(* CoDeSys 2.3.9.47 project: gym_err.prx *)
(* Libraries: TcBaseBX.lbx 10.5.06 08:50:20, TcSystemBX.lbx 11.6.12 13:56:16, standard.lbx 5.12.03 08:02:30, TcEIB.lbx 16.5.14 14:12:22, TcBABasicBX.lbx 22.7.15 15:46:56 *)

(* Task configuration *)
TASK Standard (PRIORITY := 0, INTERVAL := T#20ms);
	MAIN
END_TASK

(* Global variable list: Global_Variables *)
VAR_GLOBAL
END_VAR

VAR_GLOBAL RETAIN
	eib_gym01:							 BOOL;
	eib_gym02:							 BOOL;
	eib_training01:						 BOOL;
	eib_training02:						 BOOL;
	eib_training03	:						 BOOL;
	eib_gym_stairs_bra:					 BOOL;
	eib_pool_hall_spotlight:				 BOOL;
	eib_pool_hall_LED:					 BOOL;

	eib_pool_light:						 BOOL;
	eib_sphere_ceiling_light:				 BOOL;
	eib_sphere_light:						 BOOL;
	eib_sphere_stars_light:					 BOOL;
	eib_gym_shower01_light:				 BOOL;
	eib_gym_shower02_light:				 BOOL;
	eib_gym_WC_corridor:					 BOOL;
	eib_gym_stairs_light:					 BOOL;

	eib_gym_WC_light:					 BOOL;
	eib_training:							 BOOL;
	eib_gym:								 BOOL;

	eib_training_1column_light	:			BOOL;
	eib_pool_inwater	:					BOOL;

	eib_pool_floor_heating_pump:			BOOL := TRUE ;
	eib_gym_floor_heating_pump:			BOOL := TRUE;
	eib_vent_heating_pump:				BOOL := TRUE;
	eib_heating_pump:					BOOL := TRUE;

	eib_outside_bigBulbs:					 BOOL;
	eib_outside_pingPongTable:			 BOOL;
	eib_outside_plantsLightning:			 BOOL;
	eib_outside_smallBulbs:				 BOOL;
END_VAR

(* Global variable list: KNX *)
VAR_GLOBAL
	fb_KL6301_0:								KL6301;


	fb_gym01_send_status_ex: 					EIB_BIT_SEND_EX;
	fb_gym02_send_status_ex: 					EIB_BIT_SEND_EX;
	fb_training01_send_status_ex: 				EIB_BIT_SEND_EX;
	fb_training02_send_status_ex: 				EIB_BIT_SEND_EX;
	fb_training03_send_status_ex: 				EIB_BIT_SEND_EX;
	fb_gym_stairs_bra_send_status_ex: 			EIB_BIT_SEND_EX;
	fb_pool_hall_spotlight_send_status_ex: 		EIB_BIT_SEND_EX;
	fb_pool_hall_LED_send_status_ex: 			EIB_BIT_SEND_EX;

	fb_pool_light_send_status_ex: 				EIB_BIT_SEND_EX;
	fb_sphere_ceiling_light_send_status_ex: 		EIB_BIT_SEND_EX;
	fb_sphere_light_send_status_ex: 			EIB_BIT_SEND_EX;
	fb_sphere_stars_light_send_status_ex: 		EIB_BIT_SEND_EX;
	fb_gym_shower01_light_send_status_ex: 		EIB_BIT_SEND_EX;
	fb_gym_shower02_light_send_status_ex: 		EIB_BIT_SEND_EX;
	fb_gym_WC_corridor_send_status_ex: 		EIB_BIT_SEND_EX;
	fb_gym_stairs_light_send_status_ex: 			EIB_BIT_SEND_EX;

	fb_gym_WC_light_send_status_ex: 			EIB_BIT_SEND_EX;
	fb_training_light_send_status_ex: 			EIB_BIT_SEND_EX;
	fb_gym_light_send_status_ex: 				EIB_BIT_SEND_EX;

	fb_gym_all_send_status_ex: 				EIB_BIT_SEND_EX;
	fb_training_all_send_status_ex: 				EIB_BIT_SEND_EX;
	fb_training_1column_send_status_ex: 		EIB_BIT_SEND_EX;
	fb_pool_inwater_send_status_ex: 			EIB_BIT_SEND_EX;


	fb_outside_bigBulbs_send_status_ex:		EIB_BIT_SEND_EX;
	fb_outside_smallBulbs_send_status_ex:		EIB_BIT_SEND_EX;
	fb_outside_pingPongTable_send_status_ex:	EIB_BIT_SEND_EX;
	fb_outside_plantsLightning_send_status_ex:	EIB_BIT_SEND_EX;

	fb_pool_floor_heating_pump_send_status_ex:	EIB_BIT_SEND_EX;
	fb_gym_floor_heating_pump_send_status_ex:	EIB_BIT_SEND_EX;
	fb_vent_heating_pump_send_status_ex:		EIB_BIT_SEND_EX;
	fb_heating_pump_send_status_ex:			EIB_BIT_SEND_EX;


	fb_pool_floor_heating_pump_read:			EIB_BIT_REC ;
	fb_gym_floor_heating_pump_read:			EIB_BIT_REC ;
	fb_vent_heating_pump_read:				EIB_BIT_REC ;
	fb_heating_pump_read:					EIB_BIT_REC ;

	fb_gym01_read: 					EIB_BIT_REC;
	fb_gym02_read: 					EIB_BIT_REC;
	fb_training01_read:				EIB_BIT_REC;
	fb_training02_read:				EIB_BIT_REC;
	fb_training03_read:				EIB_BIT_REC;
	fb_gym_stairs_bra_read:			EIB_BIT_REC;
	fb_pool_hall_spotlight_read:		EIB_BIT_REC;
	fb_pool_hall_LED_read:			EIB_BIT_REC;

	fb_pool_light_read:				EIB_BIT_REC;
	fb_sphere_ceiling_light_read:		EIB_BIT_REC;
	fb_sphere_light_read:				EIB_BIT_REC;
	fb_sphere_stars_light_read:			EIB_BIT_REC;
	fb_gym_shower01_light_read:		EIB_BIT_REC;
	fb_gym_shower02_light_read:		EIB_BIT_REC;
	fb_gym_WC_corridor_read:			EIB_BIT_REC;
	fb_gym_stairs_light_read:			EIB_BIT_REC;

	fb_gym_WC_light_read:			EIB_BIT_REC;
	fb_training_light_read:				EIB_BIT_REC;
	fb_gym_light_read:				EIB_BIT_REC;
	fb_outside_bigBulbs_read:			EIB_BIT_REC;
	fb_outside_smallBulbs_read:		EIB_BIT_REC;
	fb_outside_pingPongTable_read:	EIB_BIT_REC;
	fb_outside_plantsLightning_read:	EIB_BIT_REC;

	fb_gym_all_read: 					EIB_BIT_REC;
	fb_training_all_read: 				EIB_BIT_REC;
	fb_training_1column_read: 			EIB_BIT_REC;
	fb_pool_inwater_read: 				EIB_BIT_REC;

	gym_lights					:	BOOL;


(*2/0/x*)
	pool_floor_heating_pump_adr:								EIB_GROUP_ADDR :=(MAIN:=2, SUB_MAIN:=0, NUMBER:=1);
	gym_floor_heating_pump_adr:								EIB_GROUP_ADDR :=(MAIN:=2, SUB_MAIN:=0, NUMBER:=2);
	vent_heating_pump_adr:									EIB_GROUP_ADDR :=(MAIN:=2, SUB_MAIN:=0, NUMBER:=3);
	heating_pump_adr:										EIB_GROUP_ADDR :=(MAIN:=2, SUB_MAIN:=0, NUMBER:=4);

	pool_floor_heating_pump_status_adr:						EIB_GROUP_ADDR :=(MAIN:=2, SUB_MAIN:=0, NUMBER:=101);
	gym_floor_heating_pump_status_adr:							EIB_GROUP_ADDR :=(MAIN:=2, SUB_MAIN:=0, NUMBER:=102);
	vent_heating_pump_status_adr:								EIB_GROUP_ADDR :=(MAIN:=2, SUB_MAIN:=0, NUMBER:=103);
	heating_pump_staus_adr:									EIB_GROUP_ADDR :=(MAIN:=2, SUB_MAIN:=0, NUMBER:=104);


(*2/1/x*)
	gym01_adr:												EIB_GROUP_ADDR :=(MAIN:=2, SUB_MAIN:=1, NUMBER:=1);
	gym02_adr:												EIB_GROUP_ADDR :=(MAIN:=2, SUB_MAIN:=1, NUMBER:=2);
	training01_adr:											EIB_GROUP_ADDR :=(MAIN:=2, SUB_MAIN:=1, NUMBER:=3);
	training02_adr:											EIB_GROUP_ADDR :=(MAIN:=2, SUB_MAIN:=1, NUMBER:=4);
	training03_adr:											EIB_GROUP_ADDR :=(MAIN:=2, SUB_MAIN:=1, NUMBER:=5);
	gym_stairs_bra_adr:										EIB_GROUP_ADDR :=(MAIN:=2, SUB_MAIN:=1, NUMBER:=6);
	pool_hall_spotlight_adr:									EIB_GROUP_ADDR :=(MAIN:=2, SUB_MAIN:=1, NUMBER:=7);
	pool_hall_LED_adr:										EIB_GROUP_ADDR :=(MAIN:=2, SUB_MAIN:=1, NUMBER:=8);
	pool_light_adr:											EIB_GROUP_ADDR :=(MAIN:=2, SUB_MAIN:=1, NUMBER:=9);
	sphere_ceiling_light_adr:									EIB_GROUP_ADDR :=(MAIN:=2, SUB_MAIN:=1, NUMBER:=10);
	sphere_light_adr:											EIB_GROUP_ADDR :=(MAIN:=2, SUB_MAIN:=1, NUMBER:=11);
	sphere_stars_light_adr:										EIB_GROUP_ADDR :=(MAIN:=2, SUB_MAIN:=1, NUMBER:=12);
	gym_shower01_light_adr:									EIB_GROUP_ADDR :=(MAIN:=2, SUB_MAIN:=1, NUMBER:=13);
	gym_shower02_light_adr:									EIB_GROUP_ADDR :=(MAIN:=2, SUB_MAIN:=1, NUMBER:=14);
	gym_WC_corridor_adr:										EIB_GROUP_ADDR :=(MAIN:=2, SUB_MAIN:=1, NUMBER:=15);
	gym_stairs_light_adr:										EIB_GROUP_ADDR:= (MAIN:=2, SUB_MAIN:=1, NUMBER:=16);
	gym_WC_light_adr:										EIB_GROUP_ADDR:= (MAIN:=2, SUB_MAIN:=1, NUMBER:=17);
	training_light_adr:											EIB_GROUP_ADDR:= (MAIN:=2, SUB_MAIN:=1, NUMBER:=18);
	gym_light_adr:											EIB_GROUP_ADDR:= (MAIN:=2, SUB_MAIN:=1, NUMBER:=19);
	training_1column_light_adr: 									EIB_GROUP_ADDR:= (MAIN:=2, SUB_MAIN:=1, NUMBER:=20);
	pool_inwater_adr: 											EIB_GROUP_ADDR:= (MAIN:=2, SUB_MAIN:=1, NUMBER:=21);




	outside_bigBulbs_adr	:									EIB_GROUP_ADDR:= (MAIN:=2, SUB_MAIN:=1, NUMBER:=25);
	outside_smallBulbs_adr:									EIB_GROUP_ADDR:= (MAIN:=2, SUB_MAIN:=1, NUMBER:=26);
	outside_pingpongTable_adr:								EIB_GROUP_ADDR:= (MAIN:=2, SUB_MAIN:=1, NUMBER:=27);
	outside_plantsLightning_adr:								EIB_GROUP_ADDR:= (MAIN:=2, SUB_MAIN:=1, NUMBER:=28);


	gym01_status_adr:										EIB_GROUP_ADDR :=(MAIN:=2, SUB_MAIN:=1, NUMBER:=101);
	gym02_status_adr:										EIB_GROUP_ADDR :=(MAIN:=2, SUB_MAIN:=1, NUMBER:=102);
	training01_status_adr:										EIB_GROUP_ADDR :=(MAIN:=2, SUB_MAIN:=1, NUMBER:=103);
	training02_status_adr:										EIB_GROUP_ADDR :=(MAIN:=2, SUB_MAIN:=1, NUMBER:=104);
	training03_status_adr:										EIB_GROUP_ADDR :=(MAIN:=2, SUB_MAIN:=1, NUMBER:=105);
	gym_stairs_bra_status_adr:									EIB_GROUP_ADDR :=(MAIN:=2, SUB_MAIN:=1, NUMBER:=106);
	pool_hall_spotlight_status_adr:								EIB_GROUP_ADDR :=(MAIN:=2, SUB_MAIN:=1, NUMBER:=107);
	pool_hall_LED_status_adr:									EIB_GROUP_ADDR :=(MAIN:=2, SUB_MAIN:=1, NUMBER:=108);
	pool_light_status_adr:										EIB_GROUP_ADDR :=(MAIN:=2, SUB_MAIN:=1, NUMBER:=109);
	sphere_ceiling_light_status_adr:								EIB_GROUP_ADDR :=(MAIN:=2, SUB_MAIN:=1, NUMBER:=110);
	sphere_light_status_adr:									EIB_GROUP_ADDR :=(MAIN:=2, SUB_MAIN:=1, NUMBER:=111);
	sphere_stars_light_status_adr:								EIB_GROUP_ADDR :=(MAIN:=2, SUB_MAIN:=1, NUMBER:=112);
	gym_shower01_light_status_adr:								EIB_GROUP_ADDR :=(MAIN:=2, SUB_MAIN:=1, NUMBER:=113);
	gym_shower02_light_status_adr:								EIB_GROUP_ADDR :=(MAIN:=2, SUB_MAIN:=1, NUMBER:=114);
	gym_WC_corridor_status_adr:								EIB_GROUP_ADDR :=(MAIN:=2, SUB_MAIN:=1, NUMBER:=115);
	gym_stairs_light_status_adr:								EIB_GROUP_ADDR:= (MAIN:=2, SUB_MAIN:=1, NUMBER:=116);
	gym_WC_light_status_adr:									EIB_GROUP_ADDR:= (MAIN:=2, SUB_MAIN:=1, NUMBER:=117);
	training_light_status_adr:									EIB_GROUP_ADDR:= (MAIN:=2, SUB_MAIN:=1, NUMBER:=118);
	gym_light_status_adr:										EIB_GROUP_ADDR:= (MAIN:=2, SUB_MAIN:=1, NUMBER:=119);
	training_1column_light_status_adr: 							EIB_GROUP_ADDR:= (MAIN:=2, SUB_MAIN:=1, NUMBER:=120);
	pool_inwater_status_adr: 									EIB_GROUP_ADDR:= (MAIN:=2, SUB_MAIN:=1, NUMBER:=121);



	outside_bigBulbs_status_adr	:							EIB_GROUP_ADDR:= (MAIN:=2, SUB_MAIN:=1, NUMBER:=125);
	outside_smallBulbs_status_adr:								EIB_GROUP_ADDR:= (MAIN:=2, SUB_MAIN:=1, NUMBER:=126);
	outside_pingPongTable_status_adr:							EIB_GROUP_ADDR:= (MAIN:=2, SUB_MAIN:=1, NUMBER:=127);
	outside_plantsLightning_status_adr:							EIB_GROUP_ADDR:= (MAIN:=2, SUB_MAIN:=1, NUMBER:=128);

END_VAR

(* Global variable list: main *)
VAR_GLOBAL
	dataDerevo: ARRAY[0..3] OF BYTE;
	dataDerevo_prev :ARRAY[0..3] OF BYTE;

	datafloor1: ARRAY[0..3] OF BYTE;
	datafloor1_prev :ARRAY[0..3] OF BYTE;



	ads_adr_derevo: STRING:='10.0.5.64.1.1';
	ads_adr_3floor: STRING:='10.0.5.63.1.1';
	ads_adr_1floor: STRING:='10.0.5.61.1.1';

	write_ads: ADSWRITE;

	bDarkOutside						AT%MX0.0:BOOL;


	iHour							AT%MB1:	BYTE;
	iMinute							AT%MB3:	BYTE;

	t_out							AT%MB6 :	 REAL;
	heartBeatTime : TIME		:= t#30m;

	floor1_tambur3_light				AT %MX100.0 :BOOL;
	sw_floor1_tambur3_short			AT %MX100.1 :BOOL;
	sw_floor1_tambur3_long			AT %MX100.2 :BOOL;
	m_heating_pump					AT %MX100.3 :BOOL;

END_VAR

(* Global variable list: TwinCAT_Import *)
VAR_GLOBAL (* DO NOT CHANGE THIS SHEET MANUALLY! *)

	gym01_light				AT %QX0.0:	BOOL; (*K01*)
	training03_light			AT %QX0.1:	BOOL; (*K05*)
	gym02_light				AT %QX0.2:	BOOL; (*K02*)
	gym_stairs_bra_right		AT %QX0.3:	BOOL; (*K06*)
	training01_light			AT %QX0.4:	BOOL; (*K03*)
	gym_stairs_bra_left		AT %QX0.5:	BOOL; (*K07*)
	training02_light			AT %QX0.6:	BOOL; (*K04*)
	pool_hall_spotlight		AT %QX0.7:	BOOL; (*K08*)

	pool_hall_ceiling_LED		AT %QX1.0:	BOOL; (*K09*)
	pool_light				AT %QX1.1:	BOOL; (*K13*)
	sphere_ceiling_light		AT %QX1.2:	BOOL; (*K10*)
	gym01_2_light			AT %QX1.3:	BOOL; (*K14*)
	sphere_light01			AT %QX1.4:	BOOL; (*K11*)
	gym02_2_light			AT %QX1.5:	BOOL; (*K15*)
	sphere_stars_light			AT %QX1.6:	BOOL; (*K12*)
	training01_2_light			AT %QX1.7:	BOOL; (*K16*)

	training02_2_light			AT %QX2.0:	BOOL; (*K17*)
	gym_shower02_light		AT %QX2.1:	BOOL; (*K21*)
	training03_2_light			AT %QX2.2:	BOOL; (*K18*)
	gym_WC_light			AT %QX2.3:	BOOL; (*K22*)
	gym_shower01_light		AT %QX2.4:	BOOL; (*K19*)
	gym_stairs_light			AT %QX2.5:	BOOL; (*K23*)
	gym_WC_corridor			AT %QX2.6:	BOOL; (*K20*)
	sphere_stairs_light		AT %QX2.7:	BOOL; (*K24*)

	pool_hall_LED			AT %QX3.0:	BOOL; (*K25*)
	outside_smallBulbs		AT %QX3.1:	BOOL;
	gym_cinema_TEMPORARY_light	AT %QX3.2:	BOOL; (*K26*)
	outside_bigBulbs			AT %QX3.3:	BOOL;
	Term_5_KL2408_5_Output	AT %QX3.4:	BOOL;
	outside_plantsLightning	AT %QX3.5:	BOOL;
	Term_5_KL2408_7_Output	AT %QX3.6:	BOOL;
	outside_pingPongTable	AT %QX3.7:	BOOL;

	out_5_1					AT %QX4.0:	BOOL; (**)
	fancoil_low_speed		AT %QX4.1:	BOOL; (*engineering K01*)
	out_5_3					AT %QX4.2:	BOOL; (**)
	fancoil_med_speed		AT %QX4.3:	BOOL; (*engineering K02*)
	out_5_5					AT %QX4.4:	BOOL; (**)
	fancoil_high_speed		AT %QX4.5:	BOOL; (*engineering K03*)
	out_5_7					AT %QX4.6:	BOOL; (**)
	pool_floor_heating_pump	AT %QX4.7:	BOOL; (*engineering K04*)

	heating_pump			AT %QX5.0:	BOOL; (*engineering K05*)
	storage_light				AT %QX5.1:	BOOL; (*engineering K09*)
	gym_floor_heating_pump	AT %QX5.2:	BOOL; (*engineering K06*)
	heating_room_light		AT %QX5.3:	BOOL; (*engineering K10*)
	vent_heating_pump		AT %QX5.4:	BOOL; (*engineering K07*)
	heating_storage_fan		AT %QX5.5:	BOOL; (*engineering K11*)
	out_6_7					AT %QX5.6:	BOOL; (*engineering K08*)
	pool_inwater				AT %QX5.7:	BOOL; (*engineering K12*)

	pool_small_light			AT %QX6.0:	BOOL; (**)
	cinema_AHU_mode		AT %QX6.1:	BOOL; (*1-auto*)
	out_7_3					AT %QX6.2:	BOOL; (**)
	cinema_AHU_high_speed	AT %QX6.3:	BOOL; (**)
	sphere_bra_left			AT %QX6.4:	BOOL; (**)
	cinema_AHU_med_speed	AT %QX6.5:	BOOL; (**)
	sphere_2_floor_ligh		AT %QX6.6:	BOOL; (**)
	cinema_AHU_low_speed	AT %QX6.7:	BOOL; (**)

	gym_floor_heating			AT %QX7.0:	BOOL; (**)
	garage_light_02			AT %QX7.1:	BOOL; (**)
	training_floor_heating01	AT %QX7.2:	BOOL; (**)
	garage_light_03			AT %QX7.3:	BOOL; (**)
	training_floor_heating02	AT %QX7.4:	BOOL; (**)
	distribution_board_light		AT %QX7.5:	BOOL; (**)
	garage_light_01			AT %QX7.6:	BOOL; (**)
	garage_out_light			AT %QX7.7:	BOOL; (**)

	training_AHU_high_speed	AT %QX8.0:	BOOL; (**)
	out_9_2					AT %QX8.1:	BOOL; (**)
	training_AHU_med_speed	AT %QX8.2:	BOOL; (**)
	out_9_4					AT %QX8.3:	BOOL; (**)
	training_AHU_low_speed	AT %QX8.4:	BOOL; (**)
	out_9_6					AT %QX8.5:	BOOL; (**)
	training_AHU_mode		AT %QX8.6:	BOOL; (**)
	out_9_8					AT %QX8.7:	BOOL; (**)


	sw_12_1					AT %IX0.0:	BOOL;
	sw_08_2					AT %IX0.1:	BOOL;
	sw_12_2					AT %IX0.2:	BOOL;
	Term_6_KL1408_4_Input	AT %IX0.3:	BOOL;
	sw_12_3					AT %IX0.4:	BOOL;
	sw_08_1					AT %IX0.5:	BOOL;
	sw_08_3					AT %IX0.6:	BOOL;
	sw_13_2					AT %IX0.7:	BOOL;

	sw_13_4					AT %IX1.0:	BOOL;
	sw_01_1					AT %IX1.1:	BOOL;
	sw_13_3					AT %IX1.2:	BOOL;
	sw_01_2					AT %IX1.3:	BOOL;
	sw_13_1					AT %IX1.4:	BOOL;
	sw_01_4					AT %IX1.5:	BOOL;
	Term_7_KL1408_7_Input	AT %IX1.6:	BOOL;
	sw_01_3					AT %IX1.7:	BOOL;

	sw_01_5					AT %IX2.0:	BOOL;
	sw_05_4					AT %IX2.1:	BOOL;
	sw_01_6					AT %IX2.2:	BOOL;
	sw_05_5					AT %IX2.3:	BOOL;
	sw_05_1					AT %IX2.4:	BOOL;
	sw_05_6					AT %IX2.5:	BOOL;
	sw_05_3					AT %IX2.6:	BOOL;
	sw_05_2					AT %IX2.7:	BOOL;

	sw_14_1					AT %IX3.0:	BOOL;
	sw_10_1					AT %IX3.1:	BOOL;
	sw_14_2					AT %IX3.2:	BOOL;
	sw_10_2					AT %IX3.3:	BOOL;
	sw_11_1					AT %IX3.4:	BOOL;
	sw_06_2					AT %IX3.5:	BOOL;
	sw_11_2					AT %IX3.6:	BOOL;
	sw_06_1					AT %IX3.7:	BOOL;

	sw_07_1_1				AT %IX4.0:	BOOL;
	sw_15_1_1				AT %IX4.1:	BOOL;
	sw_07_1_2				AT %IX4.2:	BOOL;
	sw_15_1_2				AT %IX4.3:	BOOL;
	sw_07_2_1				AT %IX4.4:	BOOL;
	sw_15_2_1				AT %IX4.5:	BOOL;
	sw_07_2_2				AT %IX4.6:	BOOL;
	sw_15_2_2				AT %IX4.7:	BOOL;

	sw_15_3_1				AT %IX5.0:	BOOL;
	swg_1_1					AT %IX5.1:	BOOL;
	sw_15_3_2				AT %IX5.2:	BOOL;
	swg_2_1					AT %IX5.3:	BOOL;
	swg_3_1					AT %IX5.4:	BOOL;
	swg_4_1					AT %IX5.5:	BOOL;
	swg_5_1					AT %IX5.6:	BOOL;
	Term_11_KL1408_8_Input	AT %IX5.7:	BOOL;

	Term_12_KL1408_1_Input	AT %IX6.0:	BOOL;
	Term_12_KL1408_2_Input	AT %IX6.1:	BOOL;
	Term_12_KL1408_3_Input	AT %IX6.2:	BOOL;
	Term_12_KL1408_4_Input	AT %IX6.3:	BOOL;
	Term_12_KL1408_5_Input	AT %IX6.4:	BOOL;
	Term_12_KL1408_6_Input	AT %IX6.5:	BOOL;
	Term_12_KL1408_7_Input	AT %IX6.6:	BOOL;
	Term_12_KL1408_8_Input	AT %IX6.7:	BOOL;


	KL6301_IN_0 				AT %IB100: ARRAY[1..24] OF BYTE;
	KL6301_OUT_0 			AT %QB100: ARRAY[1..24] OF BYTE;

END_VAR

(* POU MAIN, ST *)
PROGRAM MAIN
VAR
	i,j:INT;
	write:BOOL;
	heartBeat: TP;
	i1: INT;
	j1: INT;
	write1: BOOL;
	sw_12_1_short_pulse:TP;
	sw_12_1_long_pulse:TP;
	sw_12_2_short_pulse:TP;
	sw_12_2_long_pulse:TP;
	sw_08_2_short_pulse:TP;
	sw_08_2_long_pulse:TP;

	sw_09_1_short_pulse: TP;
	sw_09_1_long_pulse: TP;
	init: BOOL := TRUE;
END_VAR
heartBeat(IN:= NOT heartBeat.Q, PT:=t#5s);

EIB;
ADS_Communication;
(*Light.knx_triggers;*)
Light.switches;
Light;
Light.outsideLight;
engineering;
(*Counters;*)
write_ADSdata;
END_PROGRAM
ACTION write_ADSdata:
	sw_12_1_short_pulse(IN:= Light.fb_sw_12_1.bShortClick, pt:=t#500ms);
	sw_12_1_long_pulse(IN:= Light.fb_sw_12_1.bLongClick, pt:=t#500ms);
	sw_12_2_short_pulse(IN:= Light.fb_sw_12_2.bShortClick, pt:=t#500ms);
	sw_12_2_long_pulse(IN:= Light.fb_sw_12_2.bLongClick, pt:=t#500ms);
	sw_08_2_short_pulse(IN:= Light.fb_sw_08_3.bShortClick, pt:=t#500ms);
	sw_08_2_long_pulse(IN:= Light.fb_sw_08_3.bLongClick, pt:=t#500ms);

	sw_09_1_short_pulse(IN:= Light.fb_sw_09_1.bShortClick, pt:=t#500ms);
	sw_09_1_long_pulse(IN:= Light.fb_sw_09_1.bLongClick, pt:=t#500ms);


	datafloor1[0].0 := sw_12_1_short_pulse.Q;
	datafloor1[0].1 := sw_12_1_long_pulse.Q;
	datafloor1[0].2 := sw_12_2_short_pulse.Q;
	datafloor1[0].3 := sw_12_2_long_pulse.Q;
	datafloor1[0].4 := gym_stairs_bra_left;
	datafloor1[0].5 := sw_08_2_short_pulse.Q;
	datafloor1[0].6 := sw_08_2_long_pulse.Q;
	datafloor1[0].7 := sw_09_1_short_pulse.Q;
	datafloor1[1].0 := sw_09_1_long_pulse.Q;

FOR i:=0 TO (SIZEOF(dataDerevo))-1 DO
	IF dataDerevo[i]<>dataDerevo_prev[i]  THEN
		write:=TRUE;
		EXIT;
	ELSE
		write:=FALSE;
	END_IF
END_FOR


FOR j:=0 TO (SIZEOF(dataDerevo))-1 DO
	dataDerevo_prev[j]:=dataDerevo[j];
END_FOR

FOR i1:=0 TO (SIZEOF(dataFloor1))-1 DO
	IF dataFloor1[i1]<>dataFloor1_prev[i1]  THEN
		write1:=TRUE;
		EXIT;
	ELSE
		write1:=FALSE;
	END_IF
END_FOR


FOR j1:=0 TO (SIZEOF(dataFloor1))-1 DO
	dataFloor1_prev[j1]:=dataFloor1[j1];
END_FOR
END_ACTION

(* POU EIB, ST *)
PROGRAM EIB
VAR

	eib_send_mode_gym:INT;
	eib_send_cyclical_start_gym: BOOL;

	floors:INT;
	i:INT;
	fb_sending_floor_order:CTU;
	fb_heartbeat_timer:TON;
	fb_sending_time_frame:TOF;

	fb_start_delay:TP;


END_VAR
fb_start_delay(IN:=  SYSTEMTASKINFOARR[1].firstCycle, PT:=t#10s);

(*EIB*)
fb_heartbeat_timer(in:=NOT  fb_heartbeat_timer.Q, pt:=heartBeatTime);
fb_sending_time_frame(in:=fb_heartbeat_timer.Q, pt:=t#50ms);
fb_sending_floor_order(cu:=fb_heartbeat_timer.Q, pv:=4,reset:=fb_sending_floor_order.CV >4, CV=>floors);

IF NOT fb_start_delay.Q THEN
	eib_send_mode_gym:=2;
ELSE
	eib_send_mode_gym:=0;
	eib_send_cyclical_start_gym:=TRUE;
END_IF


CASE floors OF
1:
	eib_send_mode_gym:=2*BOOL_TO_INT(NOT (fb_sending_time_frame.Q)); (*0-manual*)
	IF fb_heartbeat_timer.Q THEN
		eib_send_cyclical_start_gym:=FALSE;
	ELSE
		eib_send_cyclical_start_gym:=TRUE;
	END_IF

	heartBeatTime := t#10m;
END_CASE


fb_KL6301_0.iMode:=1;
CASE i OF
0:	(* EIB Address 1.1.2 *)
	fb_KL6301_0.EIB_PHYS_ADDR.Area:=1;
	fb_KL6301_0.EIB_PHYS_ADDR.Line:=1;
	fb_KL6301_0.EIB_PHYS_ADDR.Device:=2;
	(* Filter 1 *)
	fb_KL6301_0.EIB_GROUP_FILTER[1].GROUP_ADDR.MAIN:=2;
	fb_KL6301_0.EIB_GROUP_FILTER[1].GROUP_ADDR.SUB_MAIN:=0;
	fb_KL6301_0.EIB_GROUP_FILTER[1].GROUP_ADDR.NUMBER:=0;
	fb_KL6301_0.EIB_GROUP_FILTER[1].GROUP_LEN:=31;
	(* Filter 2*)
	fb_KL6301_0.EIB_GROUP_FILTER[2].GROUP_ADDR.MAIN:=2;
	fb_KL6301_0.EIB_GROUP_FILTER[2].GROUP_ADDR.SUB_MAIN:=1;
	fb_KL6301_0.EIB_GROUP_FILTER[2].GROUP_ADDR.NUMBER:=0;
	fb_KL6301_0.EIB_GROUP_FILTER[2].GROUP_LEN:=31;
	(* Filter 3*)
	fb_KL6301_0.EIB_GROUP_FILTER[3].GROUP_ADDR.MAIN:=2;
	fb_KL6301_0.EIB_GROUP_FILTER[3].GROUP_ADDR.SUB_MAIN:=2;
	fb_KL6301_0.EIB_GROUP_FILTER[3].GROUP_ADDR.NUMBER:=0;
	fb_KL6301_0.EIB_GROUP_FILTER[3].GROUP_LEN:=31;
	(* Filter 4 *)
	fb_KL6301_0.EIB_GROUP_FILTER[4].GROUP_ADDR.MAIN:=2;
	fb_KL6301_0.EIB_GROUP_FILTER[4].GROUP_ADDR.SUB_MAIN:=3;
	fb_KL6301_0.EIB_GROUP_FILTER[4].GROUP_ADDR.NUMBER:=0;
	fb_KL6301_0.EIB_GROUP_FILTER[4].GROUP_LEN:=31;
	(* Filter 5*)
	fb_KL6301_0.EIB_GROUP_FILTER[5].GROUP_ADDR.MAIN:=2;
	fb_KL6301_0.EIB_GROUP_FILTER[5].GROUP_ADDR.SUB_MAIN:=4;
	fb_KL6301_0.EIB_GROUP_FILTER[5].GROUP_ADDR.NUMBER:=0;
	fb_KL6301_0.EIB_GROUP_FILTER[5].GROUP_LEN:=31;
	(* Filter 6*)
	fb_KL6301_0.EIB_GROUP_FILTER[6].GROUP_ADDR.MAIN:=2;
	fb_KL6301_0.EIB_GROUP_FILTER[6].GROUP_ADDR.SUB_MAIN:=5;
	fb_KL6301_0.EIB_GROUP_FILTER[6].GROUP_ADDR.NUMBER:=0;
	fb_KL6301_0.EIB_GROUP_FILTER[6].GROUP_LEN:=31;
	(* Filter 7*)
	fb_KL6301_0.EIB_GROUP_FILTER[7].GROUP_ADDR.MAIN:=2;
	fb_KL6301_0.EIB_GROUP_FILTER[7].GROUP_ADDR.SUB_MAIN:=6;
	fb_KL6301_0.EIB_GROUP_FILTER[7].GROUP_ADDR.NUMBER:=0;
	fb_KL6301_0.EIB_GROUP_FILTER[7].GROUP_LEN:=31;
	(* Filter 8*)
	fb_KL6301_0.EIB_GROUP_FILTER[8].GROUP_ADDR.MAIN:=1;
	fb_KL6301_0.EIB_GROUP_FILTER[8].GROUP_ADDR.SUB_MAIN:=7;
	fb_KL6301_0.EIB_GROUP_FILTER[8].GROUP_ADDR.NUMBER:=0;
	fb_KL6301_0.EIB_GROUP_FILTER[8].GROUP_LEN:=31;

	fb_KL6301_0.bActivate :=TRUE; 	(*Start EIB Functionblock*)
	IF fb_KL6301_0.bReady THEN	(*Wait until the fb is ready *)
		IF NOT fb_KL6301_0.bError THEN
			i:=1;  (* EIB functionblock is now ready to send and receive *)
		ELSE
			i:=100; (* EIB ERROR*)
		END_IF
	END_IF
1:	;
100:	;(*ERROR EIB*)
END_CASE

fb_KL6301_0(
	idx:=1,								(* for every KL6301 an other idx number
										Example KL6301 terminal 1 - idx=1 , KL6301 termnal 2 -idx=3,... max. 64 *)
	KL6301_IN:=KL6301_IN_0,				(* Terminal variable - address IN *)
	KL6301_OUT:=KL6301_OUT_0 );			(* Terminal variable - address OUT *)



gym_and_outside;
END_PROGRAM
ACTION gym_and_outside:
fb_gym01_read(
	strData_Rec:=fb_KL6301_0.str_Data_Rec,
	Group_Address:=gym01_adr,
	);
IF NOT fb_gym01_read.bDataReceive THEN
	eib_gym01 := fb_gym01_read.bData;
END_IF

fb_gym02_read(
	strData_Rec:=fb_KL6301_0.str_Data_Rec,
	Group_Address:=gym02_adr,
	);
IF NOT fb_gym02_read.bDataReceive THEN
	eib_gym02 := fb_gym02_read.bData;
END_IF

fb_gym_all_read(
	strData_Rec:=fb_KL6301_0.str_Data_Rec,
	Group_Address:=gym_light_adr,
	);
IF NOT fb_gym_all_read.bDataReceive THEN
	eib_gym := fb_gym_all_read.bData;
	eib_gym01 := fb_gym_all_read.bData;
	eib_gym02 := fb_gym_all_read.bData;
END_IF

fb_training01_read(
	strData_Rec:=fb_KL6301_0.str_Data_Rec,
	Group_Address:=training01_adr,
	);
IF NOT fb_training01_read.bDataReceive THEN
	eib_training01 := fb_training01_read.bData;
END_IF

fb_training02_read(
	strData_Rec:=fb_KL6301_0.str_Data_Rec,
	Group_Address:=training02_adr,
	);
IF NOT fb_training02_read.bDataReceive THEN
	eib_training02 := fb_training02_read.bData;
END_IF

fb_training03_read(
	strData_Rec:=fb_KL6301_0.str_Data_Rec,
	Group_Address:=training03_adr
	);
IF NOT fb_training03_read.bDataReceive THEN
	eib_training03 := fb_training03_read.bData;
END_IF

fb_training_all_read(
	strData_Rec:=fb_KL6301_0.str_Data_Rec,
	Group_Address:=training_light_adr
	);
IF NOT fb_training_all_read.bDataReceive THEN
	eib_training01 := fb_training_all_read.bData;
	eib_training02 := fb_training_all_read.bData;
	eib_training03 := fb_training_all_read.bData;
	eib_training_1column_light:= fb_training_all_read.bData;
	eib_training := fb_training_all_read.bData;
END_IF


fb_training_1column_read(
	strData_Rec:=fb_KL6301_0.str_Data_Rec,
	Group_Address:=training_1column_light_adr,
	);
IF NOT fb_training_1column_read.bDataReceive THEN
	eib_training_1column_light := fb_training_1column_read.bData;
END_IF

fb_gym_stairs_bra_read(
	strData_Rec:=fb_KL6301_0.str_Data_Rec,
	Group_Address:=gym_stairs_bra_adr,
	bData=>eib_gym_stairs_bra
	);

fb_pool_hall_spotlight_read(
	strData_Rec:=fb_KL6301_0.str_Data_Rec,
	Group_Address:=pool_hall_spotlight_adr,
	bData=>eib_pool_hall_spotlight,
	);

fb_pool_hall_LED_read(
	strData_Rec:=fb_KL6301_0.str_Data_Rec,
	Group_Address:=pool_hall_LED_adr,
	bData=>eib_pool_hall_LED
	);

fb_pool_light_read(
	strData_Rec:=fb_KL6301_0.str_Data_Rec,
	Group_Address:=pool_light_adr,
	bData=>eib_pool_light
	);

fb_pool_inwater_read(
	strData_Rec:=fb_KL6301_0.str_Data_Rec,
	Group_Address:=pool_inwater_adr,
	bData=>eib_pool_inwater
	);

fb_sphere_ceiling_light_read(
	strData_Rec:=fb_KL6301_0.str_Data_Rec,
	Group_Address:=sphere_ceiling_light_adr,
	bData=>eib_sphere_ceiling_light
	);

fb_sphere_light_read(
	strData_Rec:=fb_KL6301_0.str_Data_Rec,
	Group_Address:=sphere_light_adr,
	bData=>eib_sphere_light
	);

fb_sphere_stars_light_read(
	strData_Rec:=fb_KL6301_0.str_Data_Rec,
	Group_Address:=sphere_stars_light_adr,
	bData=>eib_sphere_stars_light
	);

fb_gym_shower01_light_read(
	strData_Rec:=fb_KL6301_0.str_Data_Rec,
	Group_Address:=gym_shower01_light_adr,
	bData=>eib_gym_shower01_light
	);

fb_gym_shower02_light_read(
	strData_Rec:=fb_KL6301_0.str_Data_Rec,
	Group_Address:=gym_shower02_light_adr,
	bData=>eib_gym_shower02_light
);

fb_gym_WC_corridor_read(
	strData_Rec:=fb_KL6301_0.str_Data_Rec,
	Group_Address:=gym_WC_corridor_adr,
	bData=>eib_gym_WC_corridor
	);

fb_gym_stairs_light_read(
	strData_Rec:=fb_KL6301_0.str_Data_Rec,
	Group_Address:=gym_stairs_bra_adr,
	bData=>eib_gym_stairs_bra
	);

fb_gym_WC_light_read(
	strData_Rec:=fb_KL6301_0.str_Data_Rec,
	Group_Address:=gym_WC_light_adr,
	bData=>eib_gym_WC_light
	);


fb_pool_floor_heating_pump_read(
	strData_Rec:=fb_KL6301_0.str_Data_Rec,
	Group_Address:=pool_floor_heating_pump_adr,
	);
IF NOT fb_pool_floor_heating_pump_read.bDataReceive THEN
	eib_pool_floor_heating_pump :=fb_pool_floor_heating_pump_read.bData;
END_IF

fb_gym_floor_heating_pump_read(
	strData_Rec:=fb_KL6301_0.str_Data_Rec,
	Group_Address:=gym_floor_heating_pump_adr,
	);
IF NOT fb_gym_floor_heating_pump_read.bDataReceive THEN
	eib_gym_floor_heating_pump :=fb_gym_floor_heating_pump_read.bData;
END_IF

fb_vent_heating_pump_read(
	strData_Rec:=fb_KL6301_0.str_Data_Rec,
	Group_Address:=vent_heating_pump_adr,
	);
IF NOT fb_vent_heating_pump_read.bDataReceive THEN
	eib_vent_heating_pump :=fb_vent_heating_pump_read.bData;
END_IF

fb_heating_pump_read(
	strData_Rec:=fb_KL6301_0.str_Data_Rec,
	Group_Address:=heating_pump_adr,
	);
IF NOT fb_heating_pump_read.bDataReceive THEN
	eib_heating_pump :=fb_heating_pump_read.bData;
END_IF

fb_outside_bigBulbs_read(
	strData_Rec:=fb_KL6301_0.str_Data_Rec,
	Group_Address:=outside_bigBulbs_adr
);
IF NOT  fb_outside_Bigbulbs_read.bDataReceive THEN
	eib_outside_bigBulbs:= fb_outside_bigBulbs_read.bdata;
END_IF

fb_outside_pingPongTable_read(
	strData_Rec:=fb_KL6301_0.str_Data_Rec,
	Group_Address:=outside_pingPongTable_adr
);
IF NOT  fb_outside_pingPongTable_read.bDataReceive THEN
	eib_outside_pingPongTable:= fb_outside_pingPongTable_read.bdata;
END_IF

fb_outside_plantsLightning_read(
	strData_Rec:=fb_KL6301_0.str_Data_Rec,
	Group_Address:=outside_plantsLightning_adr
	);
IF NOT  fb_outside_plantsLightning_read.bDataReceive THEN
	eib_outside_plantsLightning:= fb_outside_plantsLightning_read.bdata;
END_IF

fb_outside_smallBulbs_read(
	strData_Rec:=fb_KL6301_0.str_Data_Rec,
	Group_Address:=outside_smallBulbs_adr
);
IF NOT  fb_outside_smallBulbs_read.bDataReceive THEN
	eib_outside_smallBulbs:= fb_outside_smallBulbs_read.bdata;
END_IF

(*sending*)

fb_gym01_send_status_ex(
	imode:=eib_send_mode_gym,
	bStart:=eib_send_cyclical_start_gym,
	str_Rec:=fb_KL6301_0.str_Data_Rec,
	bData:=gym01_light OR gym01_2_light,
	Group_Address:=gym01_status_adr
	);

fb_gym02_send_status_ex(
	imode:=eib_send_mode_gym,
	bStart:=eib_send_cyclical_start_gym,
	str_Rec:=fb_KL6301_0.str_Data_Rec,
	bData:=gym02_light OR gym02_2_light,
	Group_Address:=gym02_status_adr
	);
fb_gym_light_send_status_ex(
	imode:=eib_send_mode_gym,
	bStart:=eib_send_cyclical_start_gym,
	str_Rec:=fb_KL6301_0.str_Data_Rec,
	bData:=gym02_2_light OR gym01_2_light,
	Group_Address:=gym_light_status_adr
	);

fb_training01_send_status_ex(
	imode:=eib_send_mode_gym,
	bStart:=eib_send_cyclical_start_gym,
	str_Rec:=fb_KL6301_0.str_Data_Rec,
	bData:=training01_light OR training01_2_light,
	Group_Address:=training01_status_adr
	);

fb_training02_send_status_ex(
	imode:=eib_send_mode_gym,
	bStart:=eib_send_cyclical_start_gym,
	str_Rec:=fb_KL6301_0.str_Data_Rec,
	bData:=training02_light OR training02_2_light,
	Group_Address:=training02_status_adr
	);
fb_gym_stairs_bra_send_status_ex(
	imode:=eib_send_mode_gym,
	bStart:=eib_send_cyclical_start_gym,
	str_Rec:=fb_KL6301_0.str_Data_Rec,
	bData:=gym_stairs_bra_left,
	Group_Address:=gym_stairs_bra_status_adr
	);
fb_training03_send_status_ex(
	imode:=eib_send_mode_gym,
	bStart:=eib_send_cyclical_start_gym,
	str_Rec:=fb_KL6301_0.str_Data_Rec,
	bData:=training03_light OR training03_2_light,
	Group_Address:=training03_status_adr
	);
fb_training_light_send_status_ex(
	imode:=eib_send_mode_gym,
	bStart:=eib_send_cyclical_start_gym,
	str_Rec:=fb_KL6301_0.str_Data_Rec,
	bData:=training01_2_light AND training03_2_light,
	Group_Address:=training_light_status_adr
	);
fb_training_1column_send_status_ex(
	imode:=eib_send_mode_gym,
	bStart:=eib_send_cyclical_start_gym,
	str_Rec:=fb_KL6301_0.str_Data_Rec,
	bData:=training01_2_light,
	Group_Address:=training_1column_light_status_adr
	);

fb_pool_hall_spotlight_send_status_ex(
	imode:=eib_send_mode_gym,
	bStart:=eib_send_cyclical_start_gym,
	str_Rec:=fb_KL6301_0.str_Data_Rec,
	bData:=pool_hall_spotlight,
	Group_Address:=pool_hall_spotlight_status_adr
	);

fb_pool_hall_LED_send_status_ex(
	imode:=eib_send_mode_gym,
	bStart:=eib_send_cyclical_start_gym,
	str_Rec:=fb_KL6301_0.str_Data_Rec,
	bData:=pool_hall_LED,
	Group_Address:=pool_hall_LED_status_adr
	);

fb_pool_light_send_status_ex(
	imode:=eib_send_mode_gym,
	bStart:=eib_send_cyclical_start_gym,
	str_Rec:=fb_KL6301_0.str_Data_Rec,
	bData:=pool_light,
	Group_Address:=pool_light_status_adr
	);

fb_pool_inwater_send_status_ex(
	imode:=eib_send_mode_gym,
	bStart:=eib_send_cyclical_start_gym,
	str_Rec:=fb_KL6301_0.str_Data_Rec,
	bData:=pool_inwater,
	Group_Address:=pool_inwater_status_adr
	);

fb_sphere_ceiling_light_send_status_ex(
	imode:=eib_send_mode_gym,
	bStart:=eib_send_cyclical_start_gym,
	str_Rec:=fb_KL6301_0.str_Data_Rec,
	bData:=sphere_ceiling_light,
	Group_Address:=sphere_ceiling_light_status_adr
	);

fb_sphere_light_send_status_ex(
	imode:=eib_send_mode_gym,
	bStart:=eib_send_cyclical_start_gym,
	str_Rec:=fb_KL6301_0.str_Data_Rec,
	bData:=sphere_light01,
	Group_Address:=sphere_light_status_adr
	);

fb_sphere_stars_light_send_status_ex(
	imode:=eib_send_mode_gym,
	bStart:=eib_send_cyclical_start_gym,
	str_Rec:=fb_KL6301_0.str_Data_Rec,
	bData:=sphere_stars_light,
	Group_Address:=sphere_stars_light_status_adr
	);

fb_gym_shower01_light_send_status_ex(
	imode:=eib_send_mode_gym,
	bStart:=eib_send_cyclical_start_gym,
	str_Rec:=fb_KL6301_0.str_Data_Rec,
	bData:=gym_shower01_light,
	Group_Address:=gym_shower01_light_status_adr
	);

fb_gym_shower02_light_send_status_ex(
	imode:=eib_send_mode_gym,
	bStart:=eib_send_cyclical_start_gym,
	str_Rec:=fb_KL6301_0.str_Data_Rec,
	bData:=gym_shower02_light,
	Group_Address:=gym_shower02_light_status_adr
	);

fb_gym_WC_corridor_send_status_ex(
	imode:=eib_send_mode_gym,
	bStart:=eib_send_cyclical_start_gym,
	str_Rec:=fb_KL6301_0.str_Data_Rec,
	bData:=gym_WC_corridor,
	Group_Address:=gym_WC_corridor_status_adr
	);

fb_gym_stairs_light_send_status_ex(
	imode:=eib_send_mode_gym,
	bStart:=eib_send_cyclical_start_gym,
	str_Rec:=fb_KL6301_0.str_Data_Rec,
	bData:=gym_stairs_light,
	Group_Address:=gym_stairs_light_status_adr
	);

fb_gym_WC_light_send_status_ex(
	imode:=eib_send_mode_gym,
	bStart:=eib_send_cyclical_start_gym,
	str_Rec:=fb_KL6301_0.str_Data_Rec,
	bData:=gym_WC_light,
	Group_Address:=gym_WC_light_status_adr
	);

fb_pool_floor_heating_pump_send_status_ex(
	imode:=eib_send_mode_gym,
	bStart:=eib_send_cyclical_start_gym,
	str_Rec:=fb_KL6301_0.str_Data_Rec,
	bData:=pool_floor_heating_pump,
	Group_Address:=pool_floor_heating_pump_status_adr
	);

fb_gym_floor_heating_pump_send_status_ex(
	imode:=eib_send_mode_gym,
	bStart:=eib_send_cyclical_start_gym,
	str_Rec:=fb_KL6301_0.str_Data_Rec,
	bData:=gym_floor_heating_pump,
	Group_Address:=gym_floor_heating_pump_status_adr
	);

fb_vent_heating_pump_send_status_ex(
	imode:=eib_send_mode_gym,
	bStart:=eib_send_cyclical_start_gym,
	str_Rec:=fb_KL6301_0.str_Data_Rec,
	bData:=vent_heating_pump,
	Group_Address:=vent_heating_pump_status_adr
	);

fb_heating_pump_send_status_ex(
	imode:=eib_send_mode_gym,
	bStart:=eib_send_cyclical_start_gym,
	str_Rec:=fb_KL6301_0.str_Data_Rec,
	bData:=heating_pump,
	Group_Address:=heating_pump_staus_adr
	);

fb_outside_bigBulbs_send_status_ex(
	imode:=eib_send_mode_gym,
	bStart:=eib_send_cyclical_start_gym,
	str_Rec:=fb_KL6301_0.str_Data_Rec,
	bData:=outside_bigBulbs,
	Group_Address:=outside_bigBulbs_status_adr
	);
fb_outside_pingPongTable_send_status_ex(
	imode:=eib_send_mode_gym,
	bStart:=eib_send_cyclical_start_gym,
	str_Rec:=fb_KL6301_0.str_Data_Rec,
	bData:=outside_pingPongTable,
	Group_Address:=outside_pingPongTable_status_adr
	);

fb_outside_plantsLightning_send_status_ex(
	imode:=eib_send_mode_gym,
	bStart:=eib_send_cyclical_start_gym,
	str_Rec:=fb_KL6301_0.str_Data_Rec,
	bData:=outside_plantsLightning,
	Group_Address:=outside_plantsLightning_status_adr
	);

fb_outside_smallBulbs_send_status_ex(
	imode:=eib_send_mode_gym,
	bStart:=eib_send_cyclical_start_gym,
	str_Rec:=fb_KL6301_0.str_Data_Rec,
	bData:=outside_smallBulbs,
	Group_Address:=outside_smallBulbs_status_adr
);
END_ACTION

(* POU ADS_Communication, CFC *)
PROGRAM ADS_Communication
VAR
	fb_DerevoADSwrite: ADSWRITE;
	fb_floor1ADSwrite: ADSWRITE;

	counter_error,counter_busy: CTU;
END_VAR
VAR (* helpers for the ST form of the networks *)
	_t21 : DWORD;
	_t23 : DWORD;
	_t42 : BOOL;
	_t50 : DWORD;
	_t52 : DWORD;
	_t56 : BOOL;
END_VAR
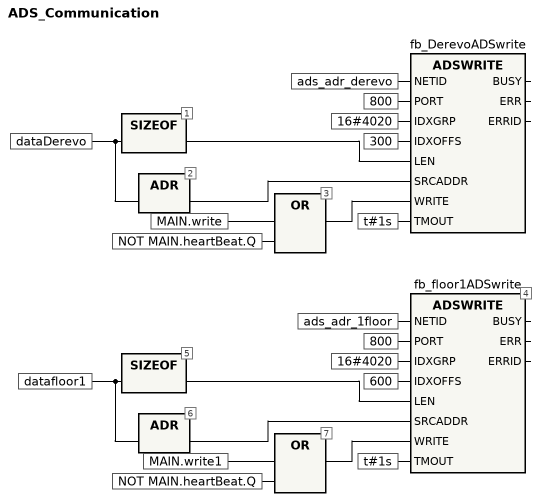
_CFC_ (* Continuous Function Chart, elements in execution order *)
#0 fb_DerevoADSwrite:ADSWRITE(NETID: ads_adr_derevo, PORT: 800, IDXGRP: 16#4020, IDXOFFS: 300, LEN: #1, SRCADDR: #2, WRITE: #3, TMOUT: t#1s)
#1 SIZEOF(dataDerevo)
#2 ADR(dataDerevo)
#3 OR(MAIN.write, NOT MAIN.heartBeat.Q)
#4 fb_floor1ADSwrite:ADSWRITE(NETID: ads_adr_1floor, PORT: 800, IDXGRP: 16#4020, IDXOFFS: 600, LEN: #5, SRCADDR: #6, WRITE: #7, TMOUT: t#1s)
#5 SIZEOF(datafloor1)
#6 ADR(datafloor1)
#7 OR(MAIN.write1, NOT MAIN.heartBeat.Q)
_END_CFC_
(* the same logic as Structured Text *)
fb_DerevoADSwrite(NETID := ads_adr_derevo, PORT := 800, IDXGRP := 16#4020, IDXOFFS := 300, LEN := _t21, SRCADDR := _t23, WRITE := _t42, TMOUT := t#1s);
_t21 := SIZEOF(dataDerevo);
_t23 := ADR(dataDerevo);
_t42 := MAIN.write OR NOT MAIN.heartBeat.Q;
fb_floor1ADSwrite(NETID := ads_adr_1floor, PORT := 800, IDXGRP := 16#4020, IDXOFFS := 600, LEN := _t50, SRCADDR := _t52, WRITE := _t56, TMOUT := t#1s);
_t50 := SIZEOF(datafloor1);
_t52 := ADR(datafloor1);
_t56 := MAIN.write1 OR NOT MAIN.heartBeat.Q;
END_PROGRAM

(* POU Light, CFC *)
PROGRAM Light
VAR
	(*switches*)


	fb_sw_01_1	:	FB_ShortLongClick;
	fb_sw_01_2	:	FB_ShortLongClick;
	fb_sw_01_3	:	FB_ShortLongClick;
	fb_sw_01_4	:	FB_ShortLongClick;
	fb_sw_01_5	:	FB_ShortLongClick;
	fb_sw_01_6	:	FB_ShortLongClick;

	fb_sw_05_1	:	FB_ShortLongClick;
	fb_sw_05_2	:	FB_ShortLongClick;
	fb_sw_05_3	:	FB_ShortLongClick;
	fb_sw_05_4	:	FB_ShortLongClick;
	fb_sw_05_5	:	FB_ShortLongClick;
	fb_sw_05_6	:	FB_ShortLongClick;
	fb_sw_06_1	:	FB_ShortLongClick;
	fb_sw_06_2	:	FB_ShortLongClick;
	fb_sw_07_1_1	:	FB_ShortLongClick;
	fb_sw_07_1_2	:	FB_ShortLongClick;
	fb_sw_08_2	:	FB_ShortLongClick;
	fb_sw_08_1	:	FB_ShortLongClick;
	fb_sw_08_3	:	FB_ShortLongClick;
	fb_sw_09_1	:	FB_ShortLongClick;
	fb_sw_10_1	:	FB_ShortLongClick;
	fb_sw_10_2	:	FB_ShortLongClick;
	fb_sw_11_1	:	FB_ShortLongClick;
	fb_sw_11_2	:	FB_ShortLongClick;
	fb_sw_12_1	:	FB_ShortLongClick;
	fb_sw_12_2	:	FB_ShortLongClick;
	fb_sw_13_1	:	FB_ShortLongClick;
	fb_sw_13_2	:	FB_ShortLongClick;
	fb_sw_13_3	:	FB_ShortLongClick;
	fb_sw_13_4	:	FB_ShortLongClick;
	fb_sw_14_1	:	FB_ShortLongClick;
	fb_sw_14_2	:	FB_ShortLongClick;

	fb_sw_15_1_1	:	FB_ShortLongClick;
	fb_sw_15_1_2	:	FB_ShortLongClick;
	fb_sw_15_2_1	:	FB_ShortLongClick;
	fb_sw_15_2_2	:	FB_ShortLongClick;
	fb_sw_15_3_1	:	FB_ShortLongClick;
	fb_sw_15_3_2	:	FB_ShortLongClick;


	longPressTimeout	:	TIME := t#500ms;

	(*Lights*)
	fb_gym01_light			: FB_Light;
	fb_gym02_light			: FB_Light;
	fb_training01_light			: FB_Light;
	fb_training02_light			: FB_Light;
	fb_training03_light			: FB_Light;
	fb_gym_stairs_bra			: FB_Light;
	fb_pool_hall_spotlight		: FB_Light;
	fb_pool_hall_LED			: FB_Light;
	fb_pool_light				: FB_Light;
	fb_sphere_ceiling_light		: FB_Light;
	fb_sphere_light			: FB_Light;
	fb_sphere_stars_light		: FB_Light;
	fb_gym_shower01_light		: FB_Light;
	fb_gym_shower02_light		: FB_Light;
	fb_gym_WC_corridor		: FB_Light;
	fb_gym_stairs_light		: FB_Light;
	fb_gym_WC_light			: FB_Light;
	fb_training_light			: FB_Light;
	fb_gym_light				: FB_Light;
	fb_training01_2_light		: FB_Light;
	fb_gym_01_2_light			: FB_Light;
	fb_gym01_2_light			: FB_Light;
	fb_pool_hall_all			: FB_Light;
	fb_cinema_temporary_light	: FB_Light;
	fb_pool_inwater			: FB_Light;


	traning_falling_edge 		:F_TRIG;
	gym_falling_edge 			:F_TRIG;

	rising_edge_eib_gym01 						:	 R_TRIG;
	rising_edge_eib_gym02 						:	 R_TRIG;
	rising_edge_eib_training01 						:	 R_TRIG;
	rising_edge_eib_training02						:	 R_TRIG;
	rising_edge_eib_training03						:	 R_TRIG;
	rising_edge_eib_gym_stairs_bra				:	 R_TRIG;
	rising_edge_eib_pool_hall_spotlight				:	 R_TRIG;
	rising_edge_eib_pool_hall_LED					:	 R_TRIG;

	rising_edge_eib_pool_light 						:	 R_TRIG;
	rising_edge_eib_sphere_ceiling_light 			:	 R_TRIG;
	rising_edge_eib_sphere_light 					:	 R_TRIG;
	rising_edge_eib_sphere_stars_light 				:	 R_TRIG;
	rising_edge_eib_gym_shower01_light			:	 R_TRIG;
	rising_edge_eib_gym_shower02_light			:	 R_TRIG;
	rising_edge_eib_gym_WC_corridor				:	 R_TRIG;
	rising_edge_eib_gym_stairs_light 				:	 R_TRIG;

	rising_edge_eib_gym_WC_light 					:	 R_TRIG;
	rising_edge_eib_training	 					:	 R_TRIG;
	rising_edge_eib_gym		 					:	 R_TRIG;

	falling_edge_eib_gym01 						:	 F_TRIG;
	falling_edge_eib_gym02 						:	 F_TRIG;
	falling_edge_eib_training01 						:	 F_TRIG;
	falling_edge_eib_training02						:	 F_TRIG;
	falling_edge_eib_training03						:	 F_TRIG;
	falling_edge_eib_gym_stairs_bra				:	 F_TRIG;
	falling_edge_eib_pool_hall_spotlight				:	 F_TRIG;
	falling_edge_eib_pool_hall_LED					:	 F_TRIG;

	falling_edge_eib_pool_light 					:	 F_TRIG;
	falling_edge_eib_sphere_ceiling_light 			:	 F_TRIG;
	falling_edge_eib_sphere_light 					:	 F_TRIG;
	falling_edge_eib_sphere_stars_light 				:	 F_TRIG;
	falling_edge_eib_gym_shower01_light			:	 F_TRIG;
	falling_edge_eib_gym_shower02_light			:	 F_TRIG;
	falling_edge_eib_gym_WC_corridor				:	 F_TRIG;
	falling_edge_eib_gym_stairs_light 				:	 F_TRIG;

	falling_edge_eib_gym_WC_light 				:	 F_TRIG;
	falling_edge_eib_training	 					:	 F_TRIG;
	falling_edge_eib_gym		 					:	 F_TRIG;

	(*timers*)
	fb_OutsideLightTimer	:TP;


	pool_all_falling_edge							: F_TRIG;
	pool_all_rising_edge							: R_TRIG;
	pool_hall_all_rising_edge						: R_TRIG;
	pool_hall_all_falling_edge						: F_TRIG;
	traning_reserved_falling_edge					: F_TRIG;

	darkOutside_rising_edge						:R_TRIG;

	darkness_correction_time_hour:INT := 20;

	pool_inwater_rising_edge						: R_TRIG;
	pool_light_rising_edge							: R_TRIG;


END_VAR
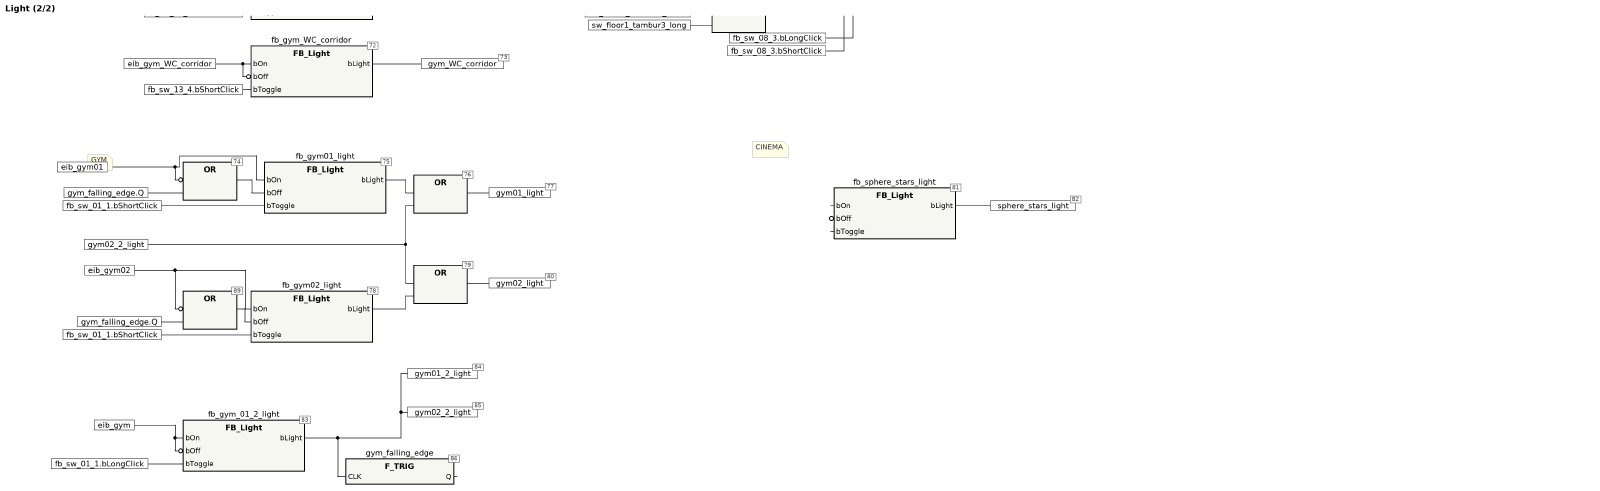
_CFC_ (* Continuous Function Chart, elements in execution order *)
(* GYM *)
(* CINEMA *)
(* SHOWER *)
(* SPHERE *)
(* POOL HALL *)
(* TRAINING ROOM *)
(* STAIRS *)
#0 OR(NOT eib_training_1column_light, traning_falling_edge.Q)
#1 fb_training01_2_light:FB_Light(bOn: eib_training_1column_light, bOff: #0, bToggle: fb_sw_08_1.bLongClick)
#2 OR(fb_sw_08_2.bLongClick, fb_sw_06_2.bLongClick, fb_sw_05_6.bLongClick)
#3 fb_training_light:FB_Light(bOn: eib_training, bOff: NOT eib_training, bToggle: #2)
#4 training02_2_light <= #3.bLight
#5 training03_2_light <= #3.bLight
#6 OR(#1.bLight, #3.bLight)
#7 training01_2_light <= #6
#8 traning_falling_edge:F_TRIG(CLK: #3.bLight)
#9 OR(traning_falling_edge.Q, traning_reserved_falling_edge.Q, NOT eib_training01)
#10 fb_training01_light:FB_Light(bOn: eib_training01, bOff: #9, bToggle: fb_sw_08_1.bShortClick)
#11 OR(#10.bLight, training01_2_light)
#12 training01_light <= #11
#13 OR(fb_sw_08_2.bShortClick, fb_sw_05_6.bShortClick, fb_sw_06_2.bShortClick)
#14 OR(NOT eib_training02, traning_falling_edge.Q)
#15 fb_training02_light:FB_Light(bOn: eib_training02, bOff: #14, bToggle: #13)
#16 traning_reserved_falling_edge:F_TRIG(CLK: #1.bLight)
#17 OR(#15.bLight, training02_2_light)
#18 training02_light <= #17
#19 OR(NOT eib_training03, traning_falling_edge.Q)
#20 fb_training03_light:FB_Light(bOn: eib_training03, bOff: #19, bToggle: #13)
#21 OR(#20.bLight, training03_2_light)
#22 training03_light <= #21
#23 OR(pool_hall_all_rising_edge.Q, eib_pool_hall_LED)
#24 OR(fb_sw_05_3.bShortClick, fb_sw_01_4.bShortClick)
#25 AND(fb_pool_hall_LED.bLight, fb_pool_hall_spotlight.bLight, pool_hall_all_falling_edge.Q)
#26 OR(NOT eib_pool_hall_LED, #25)
#27 fb_pool_hall_LED:FB_Light(bOn: #23, bOff: #26, bToggle: #24)
#28 pool_hall_ceiling_LED <= #27.bLight
#29 pool_hall_LED <= #27.bLight
#30 OR(pool_hall_all_rising_edge.Q, eib_pool_hall_spotlight)
#31 OR(NOT eib_pool_hall_spotlight, #25)
#32 OR(fb_sw_05_4.bShortClick, fb_sw_01_3.bShortClick)
#33 fb_pool_hall_spotlight:FB_Light(bOn: #30, bOff: #31, bToggle: #32)
#34 pool_hall_spotlight <= #33.bLight
#35 AND(#27.bLight, #33.bLight)
#36 pool_all_falling_edge:F_TRIG(CLK: #35)
#37 pool_all_rising_edge:R_TRIG(CLK: #35)
#38 OR(fb_sw_05_3.bLongClick, fb_sw_01_4.bLongClick, fb_sw_05_3.bLongClick, fb_sw_01_4.bLongClick)
#39 fb_pool_hall_all:FB_Light(bOn: pool_all_rising_edge.Q, bOff: pool_all_falling_edge.Q, bToggle: #38)
#40 pool_hall_all_falling_edge:F_TRIG(CLK: #39.bLight)
#41 pool_hall_all_rising_edge:R_TRIG(CLK: #39.bLight)
#42 OR(fb_sw_05_1.bLongClick, fb_sw_01_5.bLongClick, eib_pool_inwater)
#43 fb_pool_inwater:FB_Light(bOn: -, bOff: -, bToggle: #88.Q)
#44 AND(fb_sw_06_1.bLongClick, fb_sphere_light.bLight, fb_sphere_ceiling_light.bLight)
#45 pool_inwater <= #43.bLight
#46 OR(NOT eib_sphere_light, #44)
#47 fb_sphere_light:FB_Light(bOn: eib_sphere_light, bOff: #46, bToggle: fb_sw_06_1.bLongClick)
#48 sphere_light01 <= #47.bLight
#49 sphere_stairs_light <= #47.bLight
#50 fb_sphere_ceiling_light:FB_Light(bOn: eib_sphere_ceiling_light, bOff: #87, bToggle: fb_sw_06_1.bShortClick)
#51 storage_light <= #50.bLight
#52 heating_room_light <= #50.bLight
#53 OR(#47.bLight, #50.bLight)
#54 sphere_ceiling_light <= #53
#55 pool_light <= #90.bLight
#56 fb_gym_shower01_light:FB_Light(bOn: eib_gym_shower01_light, bOff: NOT eib_gym_shower01_light, bToggle: fb_sw_13_2.bShortClick)
#57 gym_shower01_light <= #56.bLight
#58 XOR(floor1_tambur3_light, gym_stairs_bra_left)
#59 OR(sw_floor1_tambur3_short, sw_floor1_tambur3_long)
#60 AND(#58, #59)
#61 OR(fb_sw_12_2.bShortClick, fb_sw_12_2.bLongClick, fb_sw_12_1.bLongClick, #60, fb_sw_08_3.bLongClick, fb_sw_08_3.bShortClick)
#62 fb_gym_stairs_bra:FB_Light(bOn: eib_gym_stairs_bra, bOff: NOT eib_gym_stairs_bra, bToggle: #61)
#63 OR(fb_sw_05_1.bShortClick, fb_sw_01_5.bShortClick)
#64 gym_stairs_bra_left <= #62.bLight
#65 gym_stairs_bra_right <= #62.bLight
#66 fb_gym_shower02_light:FB_Light(bOn: eib_gym_shower02_light, bOff: NOT eib_gym_shower02_light, bToggle: fb_sw_13_1.bShortClick)
#67 gym_shower02_light <= #66.bLight
#68 fb_gym_stairs_light:FB_Light(bOn: -, bOff: -, bToggle: -)
#69 gym_stairs_light <= #68.bLight
#70 fb_gym_WC_light:FB_Light(bOn: eib_gym_WC_light, bOff: NOT eib_gym_WC_light, bToggle: fb_sw_13_3.bShortClick)
#71 gym_WC_light <= #70.bLight
#72 fb_gym_WC_corridor:FB_Light(bOn: eib_gym_WC_corridor, bOff: NOT eib_gym_WC_corridor, bToggle: fb_sw_13_4.bShortClick)
#73 gym_WC_corridor <= #72.bLight
#74 OR(NOT eib_gym01, gym_falling_edge.Q)
#75 fb_gym01_light:FB_Light(bOn: eib_gym01, bOff: #74, bToggle: fb_sw_01_1.bShortClick)
#76 OR(#75.bLight, gym02_2_light)
#77 gym01_light <= #76
#78 fb_gym02_light:FB_Light(bOn: eib_gym02, bOff: #89, bToggle: fb_sw_01_1.bShortClick)
#79 OR(gym02_2_light, #78.bLight)
#80 gym02_light <= #79
#81 fb_sphere_stars_light:FB_Light(bOn: -, bOff: -, bToggle: -)
#82 sphere_stars_light <= #81.bLight
#83 fb_gym_01_2_light:FB_Light(bOn: eib_gym, bOff: NOT eib_gym, bToggle: fb_sw_01_1.bLongClick)
#84 gym01_2_light <= #83.bLight
#85 gym02_2_light <= #83.bLight
#86 gym_falling_edge:F_TRIG(CLK: #83.bLight)
#87 OR(NOT eib_sphere_ceiling_light, #44)
#88 pool_inwater_rising_edge:R_TRIG(CLK: #42)
#89 OR(NOT eib_gym02, gym_falling_edge.Q)
#90 fb_pool_light:FB_Light(bOn: eib_pool_light, bOff: NOT eib_pool_light, bToggle: #63)
_END_CFC_
END_PROGRAM
ACTION knx_triggers:
	rising_edge_eib_gym01 						(CLK:= eib_gym01);
	rising_edge_eib_gym02 						(CLK:= eib_gym02);
	rising_edge_eib_training01 					(CLK:= eib_training01);
	rising_edge_eib_training02						(CLK:=eib_training02 );
	rising_edge_eib_training03						(CLK:= eib_training03);
	rising_edge_eib_gym_stairs_bra				(CLK:= eib_gym_stairs_bra);
	rising_edge_eib_pool_hall_spotlight				(CLK:=eib_pool_hall_spotlight );
	rising_edge_eib_pool_hall_LED				(CLK:= eib_pool_hall_LED);

	rising_edge_eib_pool_light 					(CLK:= eib_pool_light);
	rising_edge_eib_sphere_ceiling_light 			(CLK:= eib_sphere_ceiling_light);
	rising_edge_eib_sphere_light 					(CLK:= eib_sphere_light);
	rising_edge_eib_sphere_stars_light 				(CLK:= eib_sphere_stars_light);
	rising_edge_eib_gym_shower01_light			(CLK:= eib_gym_shower01_light);
	rising_edge_eib_gym_shower02_light			(CLK:= eib_gym_shower02_light);
	rising_edge_eib_gym_WC_corridor				(CLK:= eib_gym_WC_corridor);
	rising_edge_eib_gym_stairs_light 				(CLK:= eib_gym_stairs_light);

	rising_edge_eib_gym_WC_light 				(CLK:= eib_gym_WC_light);
	rising_edge_eib_training	 					(CLK:= eib_training);
	rising_edge_eib_gym		 					(CLK:= eib_gym);

	falling_edge_eib_gym01 						(CLK:= eib_gym01);
	falling_edge_eib_gym02 						(CLK:= eib_gym02);
	falling_edge_eib_training01 					(CLK:= eib_training01);
	falling_edge_eib_training02						(CLK:=eib_training02 );
	falling_edge_eib_training03						(CLK:= eib_training03);
	falling_edge_eib_gym_stairs_bra				(CLK:= eib_gym_stairs_bra);
	falling_edge_eib_pool_hall_spotlight				(CLK:=eib_pool_hall_spotlight );
	falling_edge_eib_pool_hall_LED				(CLK:= eib_pool_hall_LED);

	falling_edge_eib_pool_light 					(CLK:= eib_pool_light);
	falling_edge_eib_sphere_ceiling_light 			(CLK:= eib_sphere_ceiling_light);
	falling_edge_eib_sphere_light 					(CLK:= eib_sphere_light);
	falling_edge_eib_sphere_stars_light 				(CLK:= eib_sphere_stars_light);
	falling_edge_eib_gym_shower01_light			(CLK:= eib_gym_shower01_light);
	falling_edge_eib_gym_shower02_light			(CLK:= eib_gym_shower02_light);
	falling_edge_eib_gym_WC_corridor				(CLK:= eib_gym_WC_corridor);
	falling_edge_eib_gym_stairs_light 				(CLK:= eib_gym_stairs_light);

	falling_edge_eib_gym_WC_light 				(CLK:= eib_gym_WC_light);
	falling_edge_eib_training	 					(CLK:= eib_training);
	falling_edge_eib_gym		 					(CLK:= eib_gym);
END_ACTION
ACTION outsideLight:
darkOutside_rising_edge(CLK:=bDarkOutside);
IF  darkOutside_rising_edge.Q  THEN
	outside_bigBulbs := TRUE;
	outside_plantsLightning:=TRUE;
	outside_smallBulbs := TRUE;

	eib_outside_bigBulbs := TRUE;
	eib_outside_plantsLightning:=TRUE;
	eib_outside_smallBulbs := TRUE;


ELSE
	outside_bigBulbs := eib_outside_bigBulbs;
	outside_plantsLightning:= eib_outside_plantsLightning;
	outside_smallBulbs := eib_outside_smallBulbs;
	outside_pingPongTable:=eib_outside_pingPongTable;

	IF iHour=0 AND iMinute>=1 AND iMinute<2 THEN
		outside_bigBulbs := FALSE;
		eib_outside_bigBulbs := FALSE;
		outside_plantsLightning:=FALSE;
		eib_outside_plantsLightning:=FALSE;
		outside_smallBulbs := FALSE;
		eib_outside_smallBulbs := FALSE;
		outside_pingPongTable := FALSE;
		eib_outside_pingPongTable := FALSE;
	END_IF

END_IF;
END_ACTION
ACTION switches:
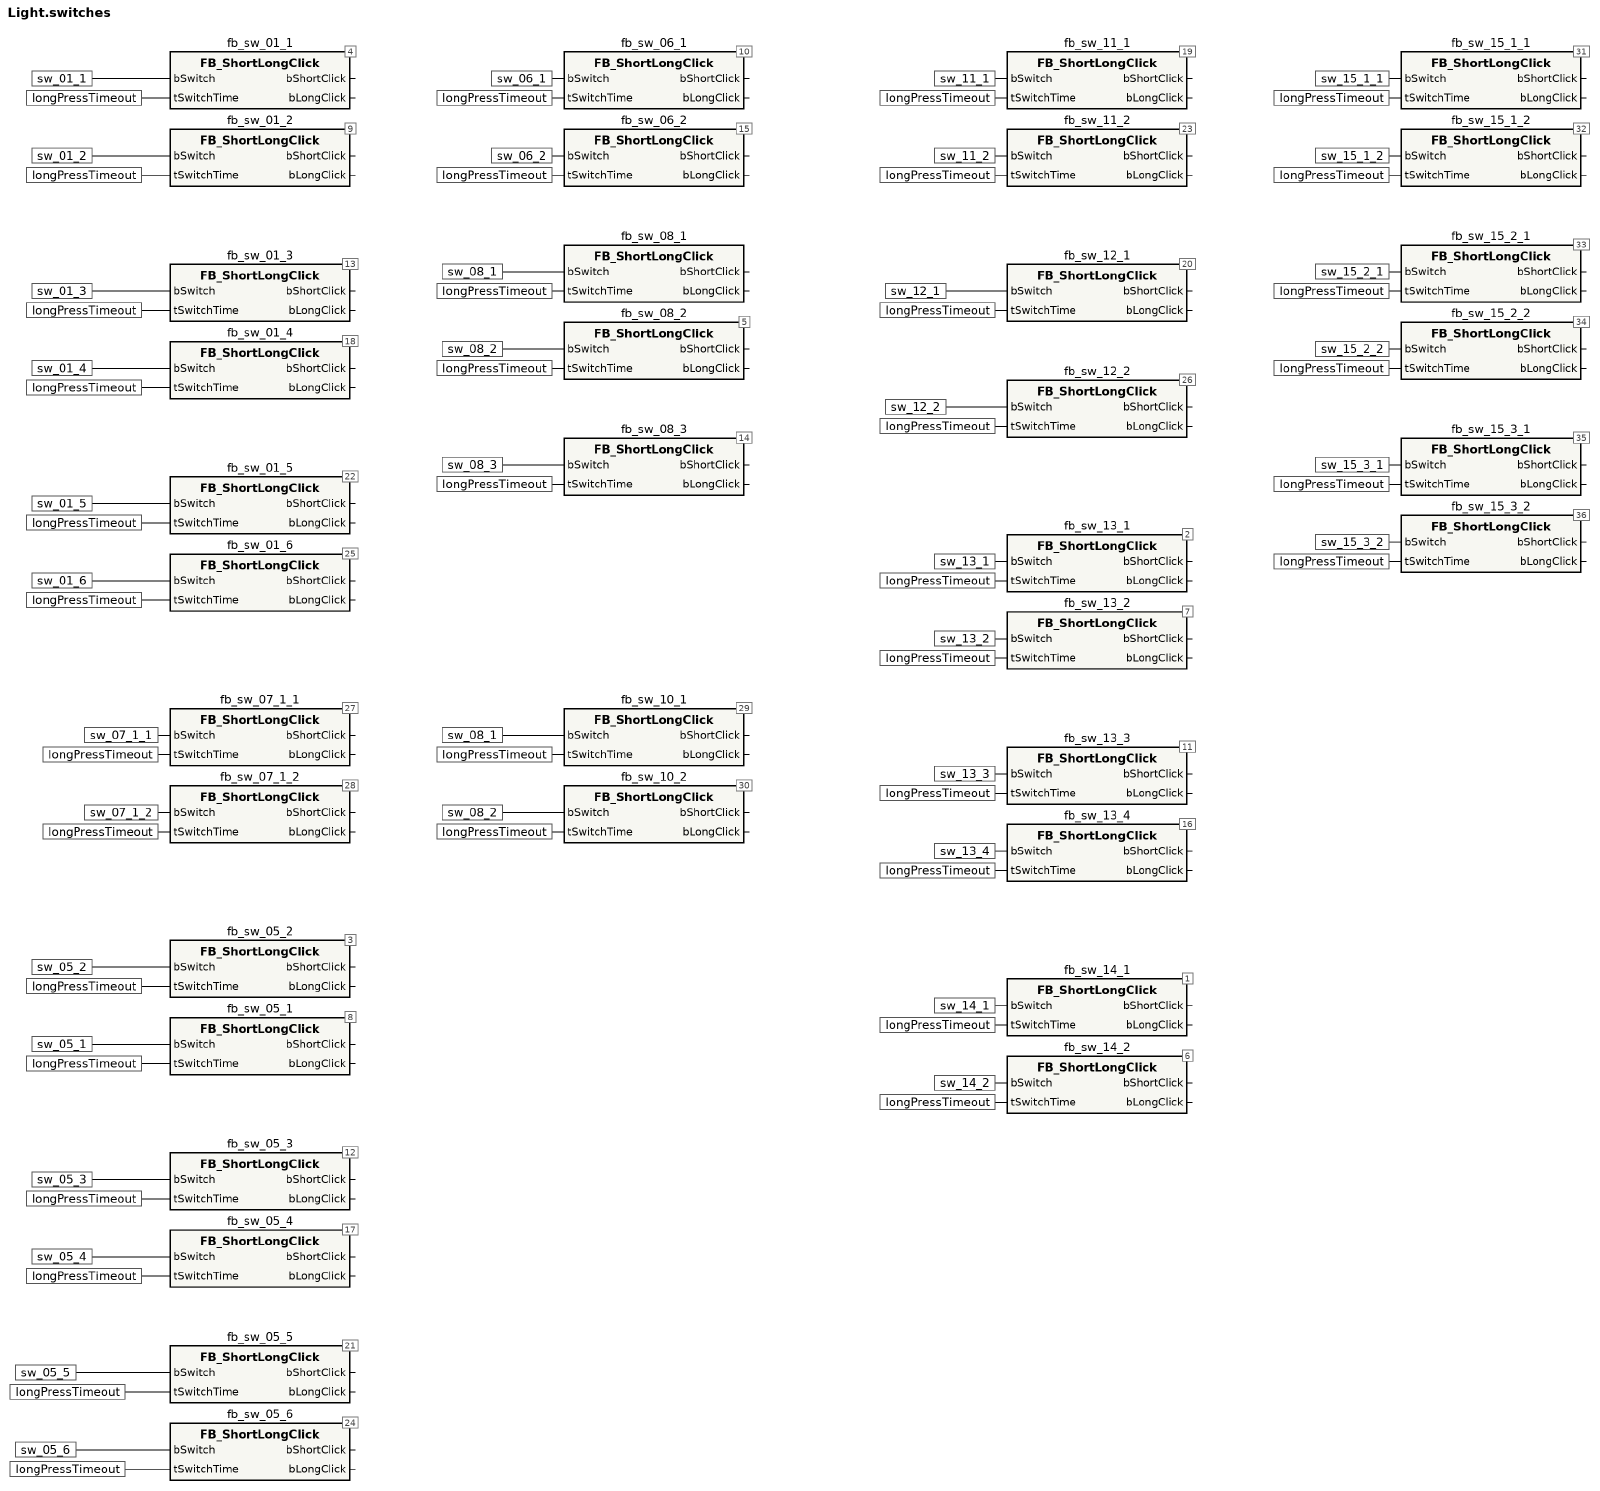
_CFC_ (* Continuous Function Chart, elements in execution order *)
#0 fb_sw_08_1:FB_ShortLongClick(bSwitch: sw_08_1, tSwitchTime: longPressTimeout)
#1 fb_sw_14_1:FB_ShortLongClick(bSwitch: sw_14_1, tSwitchTime: longPressTimeout)
#2 fb_sw_13_1:FB_ShortLongClick(bSwitch: sw_13_1, tSwitchTime: longPressTimeout)
#3 fb_sw_05_2:FB_ShortLongClick(bSwitch: sw_05_2, tSwitchTime: longPressTimeout)
#4 fb_sw_01_1:FB_ShortLongClick(bSwitch: sw_01_1, tSwitchTime: longPressTimeout)
#5 fb_sw_08_2:FB_ShortLongClick(bSwitch: sw_08_2, tSwitchTime: longPressTimeout)
#6 fb_sw_14_2:FB_ShortLongClick(bSwitch: sw_14_2, tSwitchTime: longPressTimeout)
#7 fb_sw_13_2:FB_ShortLongClick(bSwitch: sw_13_2, tSwitchTime: longPressTimeout)
#8 fb_sw_05_1:FB_ShortLongClick(bSwitch: sw_05_1, tSwitchTime: longPressTimeout)
#9 fb_sw_01_2:FB_ShortLongClick(bSwitch: sw_01_2, tSwitchTime: longPressTimeout)
#10 fb_sw_06_1:FB_ShortLongClick(bSwitch: sw_06_1, tSwitchTime: longPressTimeout)
#11 fb_sw_13_3:FB_ShortLongClick(bSwitch: sw_13_3, tSwitchTime: longPressTimeout)
#12 fb_sw_05_3:FB_ShortLongClick(bSwitch: sw_05_3, tSwitchTime: longPressTimeout)
#13 fb_sw_01_3:FB_ShortLongClick(bSwitch: sw_01_3, tSwitchTime: longPressTimeout)
#14 fb_sw_08_3:FB_ShortLongClick(bSwitch: sw_08_3, tSwitchTime: longPressTimeout)
#15 fb_sw_06_2:FB_ShortLongClick(bSwitch: sw_06_2, tSwitchTime: longPressTimeout)
#16 fb_sw_13_4:FB_ShortLongClick(bSwitch: sw_13_4, tSwitchTime: longPressTimeout)
#17 fb_sw_05_4:FB_ShortLongClick(bSwitch: sw_05_4, tSwitchTime: longPressTimeout)
#18 fb_sw_01_4:FB_ShortLongClick(bSwitch: sw_01_4, tSwitchTime: longPressTimeout)
#19 fb_sw_11_1:FB_ShortLongClick(bSwitch: sw_11_1, tSwitchTime: longPressTimeout)
#20 fb_sw_12_1:FB_ShortLongClick(bSwitch: sw_12_1, tSwitchTime: longPressTimeout)
#21 fb_sw_05_5:FB_ShortLongClick(bSwitch: sw_05_5, tSwitchTime: longPressTimeout)
#22 fb_sw_01_5:FB_ShortLongClick(bSwitch: sw_01_5, tSwitchTime: longPressTimeout)
#23 fb_sw_11_2:FB_ShortLongClick(bSwitch: sw_11_2, tSwitchTime: longPressTimeout)
#24 fb_sw_05_6:FB_ShortLongClick(bSwitch: sw_05_6, tSwitchTime: longPressTimeout)
#25 fb_sw_01_6:FB_ShortLongClick(bSwitch: sw_01_6, tSwitchTime: longPressTimeout)
#26 fb_sw_12_2:FB_ShortLongClick(bSwitch: sw_12_2, tSwitchTime: longPressTimeout)
#27 fb_sw_07_1_1:FB_ShortLongClick(bSwitch: sw_07_1_1, tSwitchTime: longPressTimeout)
#28 fb_sw_07_1_2:FB_ShortLongClick(bSwitch: sw_07_1_2, tSwitchTime: longPressTimeout)
#29 fb_sw_10_1:FB_ShortLongClick(bSwitch: sw_08_1, tSwitchTime: longPressTimeout)
#30 fb_sw_10_2:FB_ShortLongClick(bSwitch: sw_08_2, tSwitchTime: longPressTimeout)
#31 fb_sw_15_1_1:FB_ShortLongClick(bSwitch: sw_15_1_1, tSwitchTime: longPressTimeout)
#32 fb_sw_15_1_2:FB_ShortLongClick(bSwitch: sw_15_1_2, tSwitchTime: longPressTimeout)
#33 fb_sw_15_2_1:FB_ShortLongClick(bSwitch: sw_15_2_1, tSwitchTime: longPressTimeout)
#34 fb_sw_15_2_2:FB_ShortLongClick(bSwitch: sw_15_2_2, tSwitchTime: longPressTimeout)
#35 fb_sw_15_3_1:FB_ShortLongClick(bSwitch: sw_15_3_1, tSwitchTime: longPressTimeout)
#36 fb_sw_15_3_2:FB_ShortLongClick(bSwitch: sw_15_3_2, tSwitchTime: longPressTimeout)
_END_CFC_
END_ACTION

(* POU engineering, ST *)
PROGRAM engineering
VAR


END_VAR
pool_floor_heating_pump := eib_pool_floor_heating_pump;
gym_floor_heating_pump := eib_gym_floor_heating_pump;
vent_heating_pump := eib_vent_heating_pump;
heating_pump := eib_heating_pump;
END_PROGRAM

(* POU Counters, ST *)
PROGRAM Counters
VAR

	counter_6_KL1408_1_Input : CTU;

	counter_6_KL1408_3_Input	:	CTU;
	counter_6_KL1408_4_Input	:	CTU;
	counter_6_KL1408_5_Input	:	CTU;
	counter_6_KL1408_6_Input	:	CTU;

	counter_6_KL1408_8_Input	:	CTU;
	counter_7_KL1408_1_Input	:	CTU;
	counter_7_KL1408_2_Input	:	CTU;
	counter_7_KL1408_3_Input	:	CTU;
	counter_7_KL1408_4_Input	:	CTU;
	counter_7_KL1408_5_Input	:	CTU;
	counter_7_KL1408_6_Input	:	CTU;
	counter_7_KL1408_7_Input	:	CTU;
	counter_7_KL1408_8_Input	:	CTU;
	counter_8_KL1408_1_Input	:	CTU;
	counter_8_KL1408_2_Input	:	CTU;
	counter_8_KL1408_3_Input	:	CTU;
	counter_8_KL1408_4_Input	:	CTU;
	counter_8_KL1408_5_Input	:	CTU;
	counter_8_KL1408_6_Input	:	CTU;
	counter_8_KL1408_7_Input	:	CTU;
	counter_8_KL1408_8_Input	:	CTU;
	counter_9_KL1408_1_Input	:	CTU;
	counter_9_KL1408_2_Input	:	CTU;
	counter_9_KL1408_3_Input	:	CTU;
	counter_9_KL1408_4_Input	:	CTU;
	counter_9_KL1408_5_Input	:	CTU;
	counter_9_KL1408_6_Input	:	CTU;
	counter_9_KL1408_7_Input	:	CTU;
	counter_9_KL1408_8_Input	:	CTU;
	counter_10_KL1408_1_Input	:	CTU;
	counter_10_KL1408_2_Input	:	CTU;
	counter_10_KL1408_3_Input	:	CTU;
	counter_10_KL1408_4_Input	:	CTU;
	counter_10_KL1408_5_Input	:	CTU;
	counter_10_KL1408_6_Input	:	CTU;
	counter_10_KL1408_7_Input	:	CTU;
	counter_10_KL1408_8_Input	:	CTU;

	sw01 : INT;
	sw02 : INT;
	sw03 : INT;
	sw04 : INT;
	sw05 : INT;
	sw06 : INT;
	sw07 : INT;
	sw08 : INT;
	sw09 : INT;
	sw10 : INT;
	sw11 : INT;
	sw12 : INT;
	sw13 : INT;
	sw14 : INT;
	sw15 : INT;
	sw16 : INT;
	sw17 : INT;
	sw18 : INT;
	sw19 : INT;
	sw20 : INT;
	sw21 : INT;
	sw22 : INT;
	sw23 : INT;
	sw24 : INT;
	sw25 : INT;
	sw26 : INT;
	sw27 : INT;
	sw28 : INT;
	sw29 : INT;
	sw30 : INT;
	sw31 : INT;
	sw32 : INT;
	sw33 : INT;
	sw34 : INT;
	sw35 : INT;
	sw36 : INT;
	sw37 : INT;
	sw38 : INT;
	sw39 : INT;


END_VAR
	counter_6_KL1408_1_Input(CU:= Term_6_KL1408_1_Input, CV=>sw01);

	counter_6_KL1408_3_Input(CU:= Term_6_KL1408_3_Input, CV=>sw02);
	counter_6_KL1408_4_Input(CU:= Term_6_KL1408_4_Input, CV=>sw03);
	counter_6_KL1408_5_Input(CU:= Term_6_KL1408_5_Input, CV=>sw04);





	counter_7_KL1408_3_Input(CU:= Term_7_KL1408_3_Input, CV=>sw09);

	counter_7_KL1408_5_Input(CU:= Term_7_KL1408_5_Input, CV=>sw11);

	counter_7_KL1408_7_Input(CU:= Term_7_KL1408_7_Input, CV=>sw13);












	counter_9_KL1408_2_Input(CU:= Term_9_KL1408_2_Input, CV=>sw24);

	counter_9_KL1408_4_Input(CU:= Term_9_KL1408_4_Input, CV=>sw26);

	counter_9_KL1408_6_Input(CU:= Term_9_KL1408_6_Input, CV=>sw28);

	counter_9_KL1408_8_Input(CU:= Term_9_KL1408_8_Input, CV=>sw30);

	counter_10_KL1408_1_Input(CU:= Term_10_KL1408_1_Input, CV=>sw31);
	counter_10_KL1408_2_Input(CU:= Term_10_KL1408_2_Input, CV=>sw32);
	counter_10_KL1408_3_Input(CU:= Term_10_KL1408_3_Input, CV=>sw33);
	counter_10_KL1408_4_Input(CU:= Term_10_KL1408_4_Input, CV=>sw34);
	counter_10_KL1408_5_Input(CU:= Term_10_KL1408_5_Input, CV=>sw35);
	counter_10_KL1408_6_Input(CU:= Term_10_KL1408_6_Input, CV=>sw36);
	counter_10_KL1408_7_Input(CU:= Term_10_KL1408_7_Input, CV=>sw37);
	counter_10_KL1408_8_Input(CU:= Term_10_KL1408_8_Input, CV=>sw38);
END_PROGRAM
